// TIA Portal V17 export
// export: Created 2025-03-10T12:17:42.1800402Z, ExportSetting WithDefaults, DisplayName Totally Integrated Automation Portal, DisplayVersion V17 Update 8, DisplayName TIA Portal Openness, DisplayVersion V17 Update 8, DisplayName TIA Portal Version Control Interface, DisplayVersion V17, DisplayName SINAMICS Startdrive Advanced, DisplayVersion V17 SP2, DisplayName SINAMICS Startdrive G110M, G120, G120C, G120D, G120P, G115D, DisplayVersion V17 SP2, DisplayName SINAMICS Startdrive G130, G150, S120, S150, SINAMICS MV, S210, DisplayVersion V17 SP2, DisplayName STEP 7 Professional, DisplayVersion V17 Update 8, DisplayName SINUMERIK ONE STEP 7 Toolbox, DisplayVersion V17 Update 12, DisplayName SINUMERIK 840D sl STEP 7 Toolbox, DisplayVersion V17 Update 12, DisplayName STEP 7 Safety, DisplayVersion V17 Update 6, DisplayName WinCC Advanced, DisplayVersion V17 Update 8
TYPE "LBP_typeMcp310StandardOutput"
TITLE = MCP 310 image / Imagen de MCP 310 / MCP 310 Abbild
// Output image of MCP 310 / Imagen de salida de MCP 310 / Ausgangsabbild von MCP 310
// stored: IsFailsafeCompliant false
   STRUCT
      auto : Bool;
      mda : Bool;
      jog : Bool;
      singleBlock : Bool;
      spindleIncrease : Bool;
      spindle100 : Bool;
      spindleDecrease : Bool;
      cycleStop : Bool;
      teachIn : Bool;
      repos : Bool;
      refPoint : Bool;
      reset : Bool;
      spindleLeft : Bool;
      spindleStop : Bool;
      spindleRight : Bool;
      cycleStart : Bool;
      inc1 : Bool;
      inc10 : Bool;
      inc100 : Bool;
      inc1000 : Bool;
      reserved24 : Bool;
      incVar : Bool;
      feedrateStop : Bool;
      feedrateStart : Bool;
      reserved3 : Byte;
      optionalKey1 : Bool;   // KT-OUT1
      optionalKey2 : Bool;   // KT-OUT2
      optionalKey3 : Bool;   // KT-OUT3
      optionalKey4 : Bool;   // KT-OUT4
      optionalKey5 : Bool;   // KT-OUT5
      rapidTraverse : Bool;
      minus : Bool;
      plus : Bool;
      axisX : Bool;
      axisY : Bool;
      axisZ : Bool;
      axis4 : Bool;
      axis5 : Bool;
      axis6 : Bool;
      optionalKey6 : Bool;   // KT-OUT6
      customerKey16 : Bool;   // T16
      customerKey15 : Bool;   // T15
      customerKey14 : Bool;   // T14
      customerKey13 : Bool;   // T13
      mcsWcs : Bool;
      customerKey12 : Bool;   // T12
      customerKey11 : Bool;   // T11
      customerKey10 : Bool;   // T10
      customerKey9 : Bool;   // T9
      customerKey8 : Bool;   // T8
      customerKey7 : Bool;   // T7
      customerKey6 : Bool;   // T6
      customerKey5 : Bool;   // T5
      customerKey4 : Bool;   // T4
      customerKey3 : Bool;   // T3
      customerKey2 : Bool;   // T2
      customerKey1 : Bool;   // T1
   END_STRUCT;
END_TYPE
